FUNCTION_BLOCK Vehicle
  (* Standard: 61499-2 *)
  (* Version 0.1, 2015-00-24, Jin, Jin-PC *)
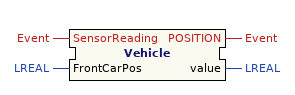
  EVENT_INPUT
    SensorReading;
  END_EVENT
  EVENT_OUTPUT
    POSITION;
  END_EVENT
  VAR_INPUT
    FrontCarPos : LREAL;
  END_VAR
  VAR_OUTPUT
    value : LREAL;
  END_VAR
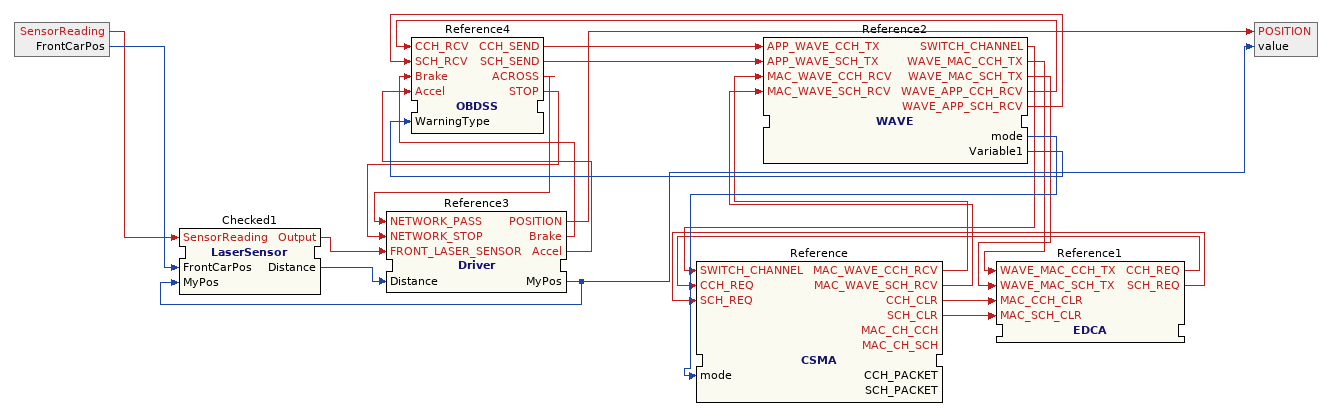
  FBS
    Reference : CSMA;
    Reference1 : EDCA;
    Reference2 : WAVE;
    Reference3 : Driver;
    Reference4 : OBDSS;
    Checked1 : LaserSensor;
  END_FBS
  EVENT_CONNECTIONS
    SensorReading TO Checked1.SensorReading;
    Reference3.POSITION TO POSITION;
    Reference.MAC_WAVE_CCH_RCV TO Reference2.MAC_WAVE_CCH_RCV;
    Reference.MAC_WAVE_SCH_RCV TO Reference2.MAC_WAVE_SCH_RCV;
    Reference.CCH_CLR TO Reference1.MAC_CCH_CLR;
    Reference.SCH_CLR TO Reference1.MAC_SCH_CLR;
    Reference1.CCH_REQ TO Reference.CCH_REQ;
    Reference1.SCH_REQ TO Reference.SCH_REQ;
    Reference2.SWITCH_CHANNEL TO Reference.SWITCH_CHANNEL;
    Reference2.WAVE_MAC_CCH_TX TO Reference1.WAVE_MAC_CCH_TX;
    Reference2.WAVE_MAC_SCH_TX TO Reference1.WAVE_MAC_SCH_TX;
    Reference2.WAVE_APP_CCH_RCV TO Reference4.CCH_RCV;
    Reference2.WAVE_APP_SCH_RCV TO Reference4.SCH_RCV;
    Reference3.Brake TO Reference4.Brake;
    Reference3.Accel TO Reference4.Accel;
    Reference4.CCH_SEND TO Reference2.APP_WAVE_CCH_TX;
    Reference4.SCH_SEND TO Reference2.APP_WAVE_SCH_TX;
    Reference4.ACROSS TO Reference3.NETWORK_PASS;
    Reference4.STOP TO Reference3.NETWORK_STOP;
    Checked1.Output TO Reference3.FRONT_LASER_SENSOR;
  END_CONNECTIONS
  DATA_CONNECTIONS
    FrontCarPos TO Checked1.FrontCarPos;
    Reference3.MyPos TO value;
    Reference2.mode TO Reference.mode;
    Reference2.Variable1 TO Reference4.WarningType;
    Reference3.MyPos TO Checked1.MyPos;
    Checked1.Distance TO Reference3.Distance;
  END_CONNECTIONS
END_FUNCTION_BLOCK
